Yaskawa INFORM job: TEST_SCAN_TRIGGER.JBI

/JOB
//NAME TEST_SCAN_TRIGGER
///FOLDERNAME TEST_JOBS
//POS
///NPOS 0,0,0,0,0,0
//ALIAS
///LVARS 0,0,2,0,0,0,0,0
LD000 SCAN_NR
LD001 USERFRAME
//INST
///DATE 2023/04/25 11:44
///ATTR SC,RW
///GROUP1 RB1
///LVARS 0,0,2,0,0,0,0,0
NOP
CALL JOB:TRIGGER_RESET
'-----
'IDs Eingeben
CALL JOB:SET_ID ARGF0 ARGF"WID"
CALL JOB:SET_ID ARGF1 ARGF"NAHT_NR"
CALL JOB:SET_ID ARGF1 ARGF"LAGE_NR"
CALL JOB:SET_ID ARGF1 ARGF"RAUPE_NR"
CALL JOB:SET_ID ARGF0 ARGF"SCHW_NR"
'-----
'Userframe setzen
SET USERFRAME 4
CALL JOB:SET_UFRAME ARGFUSERFRAME
'-----
'Scanner auswählen
SET SCAN_NR 1
'-----
'Set SCANNER TCP
CALL JOB:SET_TCPON ARGF1
TCPON TL#(1)
'-----
'Trigger Test
TIMER T=0.50
CALL JOB:LLT ARGFSCAN_NR ARGF"LASER_EIN"
TIMER T=0.50
CALL JOB:LLT ARGFSCAN_NR ARGF"TRIG_EXT"
TIMER T=0.50
CALL JOB:LLT ARGFSCAN_NR ARGF"TRIG_EIN"
TIMER T=5.00
CALL JOB:LLT ARGFSCAN_NR ARGF"TRIG_AUS"
TIMER T=0.50
CALL JOB:LLT ARGFSCAN_NR ARGF"LASER_AUS"
TIMER T=0.50
CALL JOB:LLT ARGFSCAN_NR ARGF"TRIG_INT"
'-----
'Set STANDARD TCP
CALL JOB:SET_TCPON ARGF0
TCPON TL#(0)
TCPOF
'-----
'Trigger Reset
CALL JOB:TRIGGER_RESET
END
